(* CoDeSys 2.3 export: PUMP_KD2.EXP *)

(* POU PRG/Pump_KD2, ST *)
PROGRAM Pump_KD2
VAR
	Pump : DRIVE;
	CMD_PumpRunLatch : BOOL := FALSE;

END_VAR
	(* Если активирован ручной режим управления вентилятором КД2 *)
	IF NOT KD2.PUMP.xMode_AUTO THEN
		KD2.PUMP.xCMD_RUN := (KD2.PUMP.xBtnRun OR CMD_PumpRunLatch)
									AND NOT (KD2.PUMP.xBtnStop);
	END_IF;

	CMD_PumpRunLatch := KD2.PUMP.xCMD_RUN;
END_PROGRAM
